FUNCTION F_DWORDFromBytes : DWORD
VAR_INPUT
    B3 : BYTE;
    B2 : BYTE;
    B1 : BYTE;
    B0 : BYTE;
END_VAR

F_DWORDFromBytes := SHL(SHL(SHL(BYTE_TO_DWORD(B3),8) OR BYTE_TO_DWORD(B2),8) OR BYTE_TO_DWORD(B1),8) OR BYTE_TO_DWORD(B0);

END_FUNCTION

(* stored: Version 1.1.0.1, ProductVersion 3.1.4022.18
   POU F_DWORDFromBytes: Id {c95b8ac3-4cac-4e1b-81d5-76da0d3ca853}, SpecialFunc None *)
